(* CoDeSys 2.3 library: WagoLibODP_05.lib *)
(* Libraries: SerComm.lib 27.8.09 11:23:02, Serial_Interface_01.lib 1.2.10 12:53:52, SysLibRtc.lib 5.10.04 10:37:42, SysLibTime.lib 5.10.04 10:39:34, mod_com.lib 17.5.05 08:45:18, Standard.lib 22.11.04 11:21:12, SYSLIBCALLBACK.LIB 20.4.05 11:04:48 *)

(* Global variable list: Globale_Konstanten *)
VAR_GLOBAL CONSTANT
	gcODP_uiBUFFER_SIZE :	UINT := 65000; (* Absolut size of modbus buffer 'gODP_awData' *)

	gcODP_uiOFFSET_ONLINEREAD : UINT := 2000; (* Absolut startindex of OnlineReadArea in modbus buffer 'gODP_awData' *)
	gcODP_uiOFFSET_ONLINEWRITE: UINT := 2100; (* Absolut startindex of OnlineWriteArea in modbus buffer 'gODP_awData' *)
	gcODP_uiOFFSET_ALARM: UINT := 60000; 	  (* Absolut startindex of AlarmData in modbus buffer 'gODP_awData' *)

	gcODP_uiOFFSET_HISTORY_BASE: UINT := 4000; (* Absolut startindex of HistoryData in modbus buffer 'gODP_awData' *)
 	gcODP_uiHISTORY_ITEM_SIZE  : UINT := 2000; (* Offest for each iHistoryItem in modbus buffer 'gODP_awData' *)
 	gcODP_uiHISTORY_ITEM_COUNT : UINT := 1440; (* Number of entries for each iHistoryItem to store actual values in modbus buffer 'gODP_awData' *)

	gcODP_uiMAXVAR_ONLINEREAD : UINT := 100; 	(* Maximum number of variables in 'gODP_asConfigRead'*)
	gcODP_uiMAXVAR_ONLINEWRITE: UINT := 100; 	(* Maximum number of variables in 'gODP_asConfigWrite'*)
	gcODP_uiMAXVAR_HISTORY 	  : UINT := 100; 	(* Maximum number of variables in 'gODP_asConfigHistory'*)

	gcODP_uiMAXVAR_ALARMS 	  : UINT := 128; 	(* Maximum number of variables in 'gODP_asConfigAlarms'*)
	gcODP_uiSIZE_COMPRESSEDALARMS : UINT := 8; 	(* Size of compressed representation of all alarms in (gcODP_uiMAXVAR_ALARMS/16) *)

	gcODP_uiMAXALARMLOGENTRIES: UINT := 256; 	(* Maximum number of alarm entries in 'grODP_asAlarmLog'*)

	gcODP_bMODBUS_SLAVE_ID: BYTE := 1; (* Slave-ID for ODP-Online-Data and ODP-Historical values *)
	gcODP_bMODBUS_ALARM_SLAVE_ID: BYTE := 10;  (* Slave-ID for ODP-Alarm's  *)

	gcODP_tALARMRESPONSETIMEOUT: TIME := t#30s; (* Timeout for no response received from ODP-Server *)
	gcODP_tALARMINTERVALLINIT: TIME := t#2s; (* Initial intervall for retransmission of alarms *)
END_VAR

VAR_GLOBAL
	gODP_awData : ARRAY [0..gcODP_uiBUFFER_SIZE] OF WORD; (* The central ModbusBuffer *)

	gODP_asConfigRead 	: ARRAY [0..gcODP_uiMAXVAR_ONLINEREAD] OF tODP_Config;  (* Config data for each online read variable *)
	gODP_iCountOnlineReadVars 	: INT; (* Number of configuared tags in OnlineReadArea *)
	gODP_tOnlineIntervall : TIME := t#15s; (* Intervall to update the OnlineReadArea *)

	gODP_asConfigWrite 	: ARRAY [0..gcODP_uiMAXVAR_ONLINEWRITE] OF tODP_Config; (* Config data for each online write variable *)
	gODP_iCountOnlineWriteVars	: INT; (* Number of configuared tags in OnlineWriteArea *)

	gODP_asConfigHistory: ARRAY [0..gcODP_uiMAXVAR_HISTORY] OF tODP_Config;     (* Config data for each historical variable *)
	gODP_iCountHistoryVars	: INT; (* Number of configuared tags in HistoryArea *)

	gODP_asConfigAlarms : ARRAY [0..gcODP_uiMAXVAR_ALARMS] OF tODP_Alarm;    (* Config data for each alarm variable *)
	gODP_iCountAlarms	: INT; (* Number of configuared vars in AlarmArea *)
	gODP_awCompressedAlarms	: ARRAY [0..gcODP_uiSIZE_COMPRESSEDALARMS] OF WORD; (* Compressed (bitcoded) reprasentation of all alarms *)
	gODP_tAlarmIntervall: TIME := gcODP_tALARMINTERVALLINIT; (* Current intervall for retransmission of alarms *)
END_VAR

VAR_GLOBAL RETAIN
	(* Internal "Tag" based log for the last alarms *)
	grODP_uiAlarmLogIndex : UINT; (* Position in ring buffer of the last detected alarm *)
	grODP_asAlarmLog : ARRAY [0..gcODP_uiMAXALARMLOGENTRIES] OF tODP_AlarmLog; (* Ring buffer to the last alarms *)

	(* Sendbuffer for bitcoded(compressed) alarms *)
	grODP_asAlarmSendBuffer : ARRAY [0..gcODP_uiMAXALARMLOGENTRIES] OF tODP_AlarmBuffer; (* Ring buffer of compressed alarms *)
	grODP_uiCurrentAlarms : UINT; (* In specification called "Alarmzeiger" *)
	grODP_uiTransmittedAlarms : UINT; (* In specification called "Sendezeiger" *)

	grODP_uiAlarmIncrementor : UINT; (* Used as startaddress in alarm telegrams (ODP specific feature) *)
END_VAR

(* Data type *)
TYPE tODP_Alarm :
  STRUCT
	sTagName 	: STRING(12); 		(* TagName, displayed in ODP-Config *)
	iTagId	 	: INT;		 		(* TagId of alarm, given in 'ODP_RegisterTag()' *)
	dwAddress	: DWORD; 			(* Address of variable that should be monitored *)
	wMbWordIdx 	: WORD; 			(* ModbusAddress: Position in ODP data array 'awOdpData'. Descreipted as "KENNUNG" in  ODP-Specification Values: 0..999 *)
	bMbBitIdx	: BYTE;		 		(* ModbusAddress: Position of this Alarm in 'wMbWordIdx'. Values: 0..15 *)
	eAlarmState	: tODP_AlarmState;	(* State: Comming, ACK, Going *)
	xOldValue 	: BOOL;				(* Store the last value *)
  END_STRUCT
END_TYPE

(* Data type *)
TYPE tODP_AlarmBuffer :
STRUCT
	awCompressedAlarms : ARRAY [0..gcODP_uiSIZE_COMPRESSEDALARMS] OF WORD; (* bitcoded representation of all alarms *)
	tTime 			   : tODP_Time;		(* Current time of event *)
END_STRUCT
END_TYPE

(* Data type *)
TYPE tODP_AlarmLog :
  STRUCT
	iTagId	 	: INT;		 		(* TagId of alarm, given in 'ODP_RegisterTag()' *)
	eAlarmState	: tODP_AlarmState;	(* State: Comming, ACK, Going *)
	tTime 		: tODP_Time;		(* Current time of event *)
  END_STRUCT
END_TYPE

(* Data type *)
TYPE tODP_AlarmState :
(
	eOdpAlarmNONE 	:= 0,  (* unknown *)
	eOdpAlarmCOME 	:= 1,  (* A new alarm has been detected *)
	eOdpAlarmACK 	:= 2,  (* Alarm successful send to PC-Software "ODP-Config" *)
	eOdpAlarmGONE 	:= 3   (* Alarm is gone *)
);
END_TYPE

(* Data type *)
TYPE tODP_Config :
  STRUCT
	sTagName : STRING(12); 		(* TagName, displayed in ODP-Config *)
	dwAddress: DWORD; 			(* Address of variable that should be monitored  *)
	eDataType: tODP_DataType;	(* Datatype of variable *)
	wIndex	 : WORD; 			(* Position in ODP data array 'awOdpData' *)
  END_STRUCT
END_TYPE

(* Data type *)
TYPE tODP_DataType :
(
	eOdpTypeBOOL 	:= 1,
	eOdpTypeCHAR 	:= 2,
	eOdpTypeINT8 	:= 3,
	eOdpTypeUINT8 	:= 4,
	eOdpTypeINT16 	:= 5,
	eOdpTypeUINT16 	:= 6,
	eOdpTypeINT32 	:= 7,
	eOdpTypeUINT32 	:= 8,
	eOdpTypeINT64 	:= 9,
	eOdpTypeUINT64 	:= 10,
	eOdpTypeFLOAT32 := 11,
	eOdpTypeFLOAT64 := 12,
	eOdpTypeSTRING 	:= 13,
	eOdpTypeBLOB 	:= 14
);
END_TYPE

(* Data type *)
TYPE tODP_Table :
(
	eOdpTableRead 	:= 1,
	eOdpTableWrite	:= 2,
	eOdpTableHistory:= 3,
	eOdpTableAlarm	:= 4
);
END_TYPE

(* Data type *)
TYPE tODP_Time :
  STRUCT
	bMinute : BYTE;
	bSecond : BYTE;
	bDay 	: BYTE;
	bHour 	: BYTE;
   	bYear 	: BYTE; (* Based on Year 1970 *)
	bMonth 	: BYTE;
  END_STRUCT
END_TYPE

(* POU PLC_PRG, ST *)
PROGRAM PLC_PRG
VAR
	(* ODP-Config Flag *)
	xODPInitDone : BOOL := FALSE;

	(* ODP variables to ODP-Config *)
	wReadVar_01 : WORD;
	iReadVar_02 : INT;
	uiReadVar_03: UINT;
	wMyPT100_Ch2 AT %IW1: WORD; (* Channel 2 of first analog input *)
	xMyFirstDI AT %IX2.0 : BOOL; (* Could not be monitored directly - must be mapped to helper*)
	wMyFirstDI : WORD; 	(* ODP helper variable for boolean process data *)

	(* ODP variables from ODP-Config *)
	wWriteVar_01 : WORD;
	iWriteVar_02 : INT;
	uiWriteVar_03: UINT;

	(* ODP error, alarms and messages *)
	xError_01 : BOOL; (* F1: 400V PowerSupply fails *)
	xError_02 : BOOL; (* Material buffer is empty   *)
	xError_03 : BOOL;
	xAlarm_01 : BOOL; (* Temperatur xy to high *)
	xAlarm_02 : BOOL;
	xAlarm_03 : BOOL;
	xMsg_01   : BOOL; (* Mode: "auto" -> "manual"  *)
	xMsg_02   : BOOL; (* Mode: "manual" -> "auto"  *)
	xMsg_03   : BOOL; (* Recepies: Load new        *)
	(* ModbusCommunication *)
	xConnected : BOOL;
	dwRequestCount:DWORD;
	dtLastRequest:DT;
	dwAlarmsCurrent:DWORD;
	dwAlarmsTransmitted:DWORD;
	dtLastTransmittedAlarm:DT;

END_VAR
(* Produce monitoring data *)
wReadVar_01 := wReadVar_01 +1;
iReadVar_02 := iReadVar_02 -2;
uiReadVar_03:= uiReadVar_03 +3;

(* Map boolean processdata on helper variable *)
wMyFirstDI := BOOL_TO_WORD(xMyFirstDI);

(* Start Modbus communication *)
ODP_AGENT(	EN:= TRUE,
			bCOM_PORT:= 0,		(* 0:= 873 Onboard; 1:= ServicePort; 2...n:= additional RS232 Modules 750-650 *)
			cbCOM_BAUDRATE:= BAUD_9600,
			cpCOM_PARITY:= PARITY_NO,
			csCOM_STOPBITS:= STOPBITS_1,
			cbsCOM_BYTESIZE:= BS_8,
			cfCOM_FLOW_CONTROL:= NO_FLOW_CONTROL, (* RTS_CTS; NO_FLOW_CONTROL *)
			xConnected => xConnected,
			dwRequestCount=> dwRequestCount,
			dtLastRequest=> dtLastRequest,
			dwAlarmsCurrent=> dwAlarmsCurrent,
			dwAlarmsTransmitted=> dwAlarmsTransmitted,
			dtLastTransmittedAlarm=> dtLastTransmittedAlarm);

(* Config ODP-Server *)
IF NOT xODPInitDone THEN
	(* Init ODP-Configblock *)
	ODP_InitOdpConfig('MyODPLogger', t#15s);
	(* Register variables of OnlineReadArea *)
	ODP_RegisterTag(eOdpTableRead, 'wReadVar_01', ADR(PLC_PRG.wReadVar_01), eOdpTypeUINT16);
	ODP_RegisterTag(eOdpTableRead, 'iReadVar_02', ADR(PLC_PRG.iReadVar_02), eOdpTypeINT16);
	ODP_RegisterTag(eOdpTableRead, 'uiReadVar_03', ADR(PLC_PRG.uiReadVar_03), eOdpTypeUINT16);
	ODP_RegisterTag(eOdpTableRead, 'myPT100_CH2', ADR(PLC_PRG.wMyPT100_Ch2), eOdpTypeUINT16);
	ODP_RegisterTag(eOdpTableRead, 'wMyFirstDI', ADR(PLC_PRG.wMyFirstDI), eOdpTypeUINT16);
	(* Register variables of OnlineWriteArea *)
	ODP_RegisterTag(eOdpTableWrite, 'wWriteVar_01', ADR(PLC_PRG.wWriteVar_01), eOdpTypeUINT16);
	ODP_RegisterTag(eOdpTableWrite, 'iWriteVar_02', ADR(PLC_PRG.iWriteVar_02), eOdpTypeINT16);
	ODP_RegisterTag(eOdpTableWrite, 'uiWriteVar_03', ADR(PLC_PRG.uiWriteVar_03), eOdpTypeUINT16);
	(* Register variables of HistoryArea *)
	ODP_RegisterTag(eOdpTableHistory, 'wReadVar_01', ADR(PLC_PRG.wReadVar_01), eOdpTypeUINT16);
	ODP_RegisterTag(eOdpTableHistory, 'iReadVar_02', ADR(PLC_PRG.iReadVar_02), eOdpTypeINT16);
	(* Register Alarm(SAM's) *)
	ODP_RegisterTag(eOdpTableAlarm, 'xError_01', ADR(PLC_PRG.xError_01), eOdpTypeBOOL);
	ODP_RegisterTag(eOdpTableAlarm, 'xError_02', ADR(PLC_PRG.xError_02), eOdpTypeBOOL);
	ODP_RegisterTag(eOdpTableAlarm, 'xError_03', ADR(PLC_PRG.xError_03), eOdpTypeBOOL);
	ODP_RegisterTag(eOdpTableAlarm, 'xAlarm_01', ADR(PLC_PRG.xAlarm_01), eOdpTypeBOOL);
	ODP_RegisterTag(eOdpTableAlarm, 'xAlarm_02', ADR(PLC_PRG.xAlarm_02), eOdpTypeBOOL);
	ODP_RegisterTag(eOdpTableAlarm, 'xAlarm_03', ADR(PLC_PRG.xAlarm_03), eOdpTypeBOOL);
	ODP_RegisterTag(eOdpTableAlarm, 'xMsg_01', ADR(PLC_PRG.xMsg_01), eOdpTypeBOOL);
	ODP_RegisterTag(eOdpTableAlarm, 'xMsg_02', ADR(PLC_PRG.xMsg_02), eOdpTypeBOOL);
	ODP_RegisterTag(eOdpTableAlarm, 'xMsg_03', ADR(PLC_PRG.xMsg_03), eOdpTypeBOOL);
	xODPInitDone := TRUE;
END_IF
END_PROGRAM

(* POU ODP_AGENT, ST *)
PROGRAM ODP_AGENT
(* This program work as conterpart for datalogger "ODP" from company VIDEC.
It waits for ODP-Request on serial port (Modbus_RTU).
In addition this program can send alarm telegrams.
*)
VAR_INPUT
	EN					:	BOOL := TRUE;
	bCOM_PORT			:	BYTE				:= 0; (* RS232 OnBoard 750-873 *)
	cbCOM_BAUDRATE		:	COM_BAUDRATE 		:= BAUD_9600;
	cpCOM_PARITY		:	COM_PARITY 			:= PARITY_NO;
	csCOM_STOPBITS		:	COM_STOPBITS 		:= STOPBITS_1;
	cbsCOM_BYTESIZE		:	COM_BYTESIZE 		:= BS_8;
	cfCOM_FLOW_CONTROL	:	COM_FLOW_CONTROL 	:= NO_FLOW_CONTROL ;
END_VAR
VAR_OUTPUT
	(* Online/Historic-Data*)
	xConnected :	BOOL; (* ODP-Server is connected *)
	dwRequestCount: DWORD; (* Number of received Modbus-Requests from ODP-Server *)
	dtLastRequest : DT; (* Timestamp of last received modbus request from ODP-Server*)
	(* Alarms *)
	dwAlarmsCurrent : DWORD; (* Number of local detected alarms  *)
	dwAlarmsTransmitted : DWORD; (* Number of transmitted alarms *)
	dtLastTransmittedAlarm : DT; (* Timestamp of last succesful tranmitted alarm *)
END_VAR
VAR
	(* ODP --------------------------------*)
	tCurTime 	: tODP_Time;

	xUpdateOdpWriteAreaRequired : BOOL; (* Update WriteArea after each modbus write access *)
	oTonRead 	: TON; (* Timer to update ReadArea with fresh values *)

	xSendAlarm	: BOOL; (* Flag to send an alarm to PC-Software "ODP-Config". Reset after receiving succesful acknoledge *)
	oTonAlarmResponseTimeout : TON; (* Timer to check if server acknoledge alarm within given time *)
	oTonAlarmIntervall	: TON; (* ODP: Intervall timer for minimal gap between two alarm telegrams *)

	(* ODP-Historic data *)
	bLastMinute : BYTE; (* Used to implement the intervall for writing historical data *)
	wState : WORD; (* Used in statemashiene to clear all historical data in seperate plc cycles *)
	uiCurrent : UINT; (* Index of a historical variable, used to iterate along all historical variables *)

	(* Modbus WatchDog ---------------------*)
	oTonWatchDog : TON; (* Timer to check if PC-Software "ODP-Config" is connected *)


	(* Serial-Interface --------------------*)
	oComPort		: SERIAL_INTERFACE;
	ReceiveBuffer	: typRING_BUFFER;
	RecBufferSize   : INT; (* Size member 'data' of bytes  *)
	abSendBuffer	: ARRAY[0..512] OF BYTE;
	iBytesToSend	: INT;  (* Number of bytes that should be send *)
	SendActive		: BOOL;
	xSendActiveOld  : BOOL;
	xReset			: BOOL;
	RecBufferOldIdx	: INT; (* Begin of next telegram in ringbuffer *)
	helpIdx 		: INT;
	iTo				: INT; (* Number of bytes to process *)
	oTonSendWait 	: TON; (* Detect falling edge of xSendActive and wait to make shure all data are transmitted *)
	xSendWait 		: BOOL;

	(* Local-Modbus-Slave -------------------*)
	SlaveId			: BYTE; (* received SlaveAddress from remote modbus master *)
	FunctionCode	: BYTE; (* received FunctionCode from remote modbus master *)
	UnitId			: BYTE;
	StartAddress	: WORD;
	NumberOfPoints	: WORD;

	LocalByte		: BYTE;
	BitCount		: BYTE;
	Mask			: BYTE;

	xSendResponse	: BOOL;
	ErrorCode		: BYTE;

	xIllegalFunctionCode: BOOL; (* Flag: Indicates the receiving of an unsupported or unknown FunctionCode *)

	abSlaveResponse	: ARRAY[0..512] OF BYTE; (* Buffer to build the response of the local Modbus-Slave *)
	iSlaveResponseLength: INT; (* Number of bytes that should be send *)
	iSlaveRequestLength : INT; (* Length of received bytes *)

	(* Local-Modbus-Master-----------------*)
	abMasterRequest		: ARRAY[0..125] OF BYTE; (* Buffer to build the Request of the local Modbus-Master *)
	xSendRequest		: BOOL; (* Flag to send one modbus-request to PC-Software "ODP-Config". Reset direct after transmission *)
	abMasterResponse	: ARRAY[0..19] OF BYTE; (* Buffer to process the Response from the remote Modbus-Master *)

	(* CRC16 Check ------------------------*)
	CALC_CRC			:	CRC16;  (* Function block to calculate CRC16 *)
	CRC_RTU				:	WORD;

	(* Little Helpers ---------------------*)
	i	: 	INT;
	wHelp :	WORD; (* *)

END_VAR
(* ODP: Get current time from RTC *)
tCurTime := ODP_GetTime(); (* Read current time from RTC *)

(* Update ODP-Config block (at index 8) each cycle *)
ODP_UpdateConfigArea(); (* Also update local RTC, when requested by PC-Software "ODP-Config" indicated by TRUE (at index 17) *)

(* Clear all historical data if requested *)
CASE wState OF
0: (* IDLE - Wait for something to do *)
	IF gODP_awData[37] = 16#0001 THEN
		uiCurrent := 0; (* Set Index to the first HistVar *)
		wState := 10; (* Go Ahead *)
	END_IF

10: (* Check if all historical data are reset to "INVALID_VALUE" *)
	IF uiCurrent < gODP_iCountHistoryVars THEN
		(* There are more HistVars to reset *)
		wState := 20; (* Go Ahead *)
	ELSE
		(* All HistVars are reseted *)
		gODP_awData[37] := 16#0000;
		wState := 0; (* Done *)
	END_IF

20: (* Overwrite all historical data of current HistVar with "INVALID_VALUE" *)
	FOR i:=0 TO gcODP_uiHISTORY_ITEM_COUNT-1 DO
		gODP_awData[gODP_asConfigHistory[uiCurrent].wIndex] := gODP_awData[36];
	END_FOR
	(* Set index to next HistVar *)
	uiCurrent := uiCurrent +1;
	wState := 10; (* Go Ahead *)
END_CASE

(* Check current values of all configurated alarms *)
ODP_CheckAlarms(tCurTime);

(* Check if an alarm have to be send to PC-Software "ODP-Config" *)
(* ODP: Intervall timer for minimal gap between two alarm telegrams *)
oTonAlarmIntervall(IN:=(NOT xSendAlarm), PT:= gODP_tAlarmIntervall);
IF oTonAlarmIntervall.Q THEN
	IF grODP_uiCurrentAlarms <> grODP_uiTransmittedAlarms THEN
		(* ALARM DETECTED: Send modbus request to PC-Software "ODP-Config" *)
		xSendAlarm := TRUE; (* Flag to send an alarm to PC-Software "ODP-Config". Reset after receiving succesful acknoledge *)
		xSendRequest := TRUE; (* Flag to send one modbus-request to PC-Software "ODP-Config". Reset direct after transmission *)
	END_IF
END_IF

(* Check if ODP-Server acknoledge alarm within given timeout *)
oTonAlarmResponseTimeout(IN:=xSendAlarm, PT:=gcODP_tALARMRESPONSETIMEOUT);
IF oTonAlarmResponseTimeout.Q THEN
	(* We do not receive the alarm acknoledge *)
	oTonAlarmResponseTimeout(IN:=FALSE); (* Reset timer *)
	gODP_tAlarmIntervall := gODP_tAlarmIntervall * 2; (* Increment retransmission intervall by factor 2 *)
	xSendAlarm := FALSE;
END_IF

(* Copy to output *)
dwAlarmsCurrent := grODP_uiCurrentAlarms;
dwAlarmsTransmitted := grODP_uiTransmittedAlarms;

(* ODP: Update historical data area*)
IF tCurTime.bMinute <> bLastMinute THEN
	bLastMinute := tCurTime.bMinute;
	ODP_UpdateHistory(tCurTime); (* Write current values to history *)
END_IF

(* ODP: Update OnlineWriteArea after each modbus write access *)
IF xUpdateOdpWriteAreaRequired THEN
	xUpdateOdpWriteAreaRequired := FALSE;
	ODP_UpdateOnlineWriteArea();
END_IF

(* ODP: Update OnlineReadArea with fresh values *)
oTonRead(IN:=TRUE, PT:= gODP_tOnlineIntervall);
IF oTonRead.Q THEN
	oTonRead(IN:=FALSE);
	ODP_UpdateOnlineReadArea();
END_IF

(* ODP: WatchDog to check connection with remote modbus master  *)
oTonWatchDog(IN:=TRUE, PT:= (gODP_tOnlineIntervall *8));
IF oTonWatchDog.Q THEN
	xConnected:= FALSE;
END_IF

(* Serial-Interface: Main -----------------------------*)
oComPort(	xOPEN_COM_PORT 	:= EN,
			bCOM_PORT_NR	:= bCOM_PORT,
			cbBAUDRATE		:= cbCOM_BAUDRATE,
			cpPARITY		:= cpCOM_PARITY,
			csSTOPBITS		:= csCOM_STOPBITS,
			cbsBYTESIZE		:= cbsCOM_BYTESIZE,
			cfFLOW_CONTROL	:= cfCOM_FLOW_CONTROL,
			iBYTES_TO_SEND	:= iBytesToSend,
			ptSEND_BUFFER	:= ADR(abSendBuffer[0]),
			xSTART_SEND		:= SendActive,
			utRECEIVE_BUFFER:= ReceiveBuffer,
			xINIT			:= xReset);

(* Detect falling edge of SendActive and wait to make shure all data are transmitted *)
IF (NOT SendActive) AND xSendActiveOld THEN
	oTonSendWait(IN:=FALSE);
END_IF
xSendActiveOld := SendActive;
oTonSendWait(IN:=TRUE , PT:= t#50ms);

IF (NOT SendActive) AND (oTonSendWait.Q) THEN
	(* Serial-Interface: Check ReceiveBuffer for something to do ------*)
	IF ReceiveBuffer.Index <> RecBufferOldIdx THEN
		RecBufferSize := SIZEOF(ReceiveBuffer.Data);
		(* Calculate number of received bytes  *)
		iTo	:= ReceiveBuffer.Index - RecBufferOldIdx ;
		(* Check if telegram exceed border of ringbuffer *)
		IF iTo < 0 THEN
			iTo := iTo + RecBufferSize;
		END_IF;
		(* Check if minimal telegram length is received *)
		IF iTo <= 4 THEN
			(************************************************************)
			RETURN;(*******  MINIMAL TELEGRAM LENGTH NOT REACHED ********)
			(************************************************************)
		ELSE (* iTo <= 4 *)
			(* Check Modbus-Slave-Address to obtain if telegram is a 'Modbus-Slave-Response' or a 'Modbus-Master-Request' *)
			SlaveId := ReceiveBuffer.Data[RecBufferOldIdx]; (* store Slaveaddress *)
			FunctionCode := ReceiveBuffer.Data[(RecBufferOldIdx+1) MOD RecBufferSize];	(* store FunctionCode *)

			IF SlaveId = gcODP_bMODBUS_ALARM_SLAVE_ID THEN (* -----  Telegram is a Modbus-Slave-Response  ------------------------*)
				(* Check Exceptionbit in field "FUNCTIONCODE" is set to recognise if successful or not *)
				IF ( FunctionCode AND 16#80) <> 0 THEN
					(* Sending "Alarm" to ODP-Server fails - retransmission is done by timeout *)
					RecBufferOldIdx := (RecBufferOldIdx +5) MOD RecBufferSize; (* Length of modbus execption telegram *)
					(* Reset flag for send alarm to ODP-Server *)
					xSendAlarm := FALSE;
					(* Increment Sendezeiger *)
					grODP_uiTransmittedAlarms := (grODP_uiTransmittedAlarms +1) MOD gcODP_uiMAXALARMLOGENTRIES;
				ELSE (* ( FunctionCode AND 16#80) <> 0 *)
					(* Sending "Alarm" to ODP-Server successful executed *)
					IF iTo >=8 THEN (* Wait until complied telegram of 8 bytes received *)
						(* Copy telegram data into 'abMasterResponse'*)
						FOR i:=0 TO iTo DO
							helpIdx := (RecBufferOldIdx + i) MOD RecBufferSize;
							abMasterResponse[i] :=  ReceiveBuffer.Data[ helpIdx ];
						END_FOR;
						(* Alarm successful transmitted, mark Alarm job as done in alarmlog *)
						ODP_UpdateAlarmLog(	0,
											eOdpAlarmACK,
											tCurTime);
						(* Set alarm transfer intervall to initial time *)
			    		gODP_tAlarmIntervall := gcODP_tALARMINTERVALLINIT;
						(* Set readpointer to the next modbus header *)
						RecBufferOldIdx := (RecBufferOldIdx +8) MOD RecBufferSize;
						(* Reset flag for send alarm to ODP-Server *)
						xSendAlarm := FALSE;
						(* Increment Sendezeiger *)
						grODP_uiTransmittedAlarms := (grODP_uiTransmittedAlarms +1) MOD gcODP_uiMAXALARMLOGENTRIES;
						dtLastTransmittedAlarm := SysRtcGetTime(TRUE);
					END_IF;
				END_IF

			ELSE (* ----- Telegram is a Modbus-Master-Request -------------------------------------------------*)
				(* Check FunctionCode *)
				CASE Functioncode OF

				16#03, (* FC3: Read Holding Registers 	*)
				16#04: (* FC4: Read Input Registers 	*)
					iSlaveRequestLength := 8;
					IF iTo >= iSlaveRequestLength THEN
						(* Check SlaveId against local SlaveAddress *)
						IF SlaveId <> gcODP_bMODBUS_SLAVE_ID THEN
							(* Ignore received telegram, just set readpointer to the next modbus header *)
							RecBufferOldIdx := (RecBufferOldIdx +iSlaveRequestLength) MOD RecBufferSize;
						ELSE
							(* Calculate CRC of modbus request from remote modbus master *)
							CALC_CRC(INPUT:=16#00, EN:=FALSE);
							FOR i := 0 TO 5 DO
								CALC_CRC(INPUT:=ReceiveBuffer.Data[(RecBufferOldIdx +i) MOD RecBufferSize], EN:=TRUE);
							END_FOR
							CRC_RTU := (ReceiveBuffer.Data[(RecBufferOldIdx+6) MOD RecBufferSize] * 16#0100)
										OR ReceiveBuffer.Data[(RecBufferOldIdx+7) MOD RecBufferSize];
							(* Check CRC *)
							IF CRC_RTU <> CALC_CRC.CRC THEN
								(* Send modbusexecption response to remote modbus master *)
								abSlaveResponse[0]:= SlaveId;  				(* Copy Slaveaddress into response *)
								abSlaveResponse[1]:= FunctionCode OR 16#80;	(* Copy FunctionCode into response and set ExceptionFlag*)
								abSlaveResponse[2]:= 16#03;	 				(* ILLEGAL DATA VALUE *)
								iSlaveResponseLength := 3;
								xSendResponse := TRUE; (***********************************)
							ELSE
								StartAddress := (ReceiveBuffer.Data[(RecBufferOldIdx+2)MOD RecBufferSize] * 16#0100)
												OR ReceiveBuffer.Data[(RecBufferOldIdx+3)MOD RecBufferSize];
								NumberOfPoints := (ReceiveBuffer.Data[(RecBufferOldIdx+4)MOD RecBufferSize] * 16#0100)
												OR ReceiveBuffer.Data[(RecBufferOldIdx+5)MOD RecBufferSize];
								(* Check modbus start address *)
								IF (StartAddress + NumberOfPoints) >= (SIZEOF(gODP_awData) /2) THEN
									(* Send modbusexecption response to remote modbus master *)
									abSlaveResponse[0]:= SlaveId;  				(* Copy SlaveAddress into response *)
									abSlaveResponse[1]:= FunctionCode OR 16#80;	(* Copy FunctionCode into response and set ExceptionFlag*)
									abSlaveResponse[2]:= 16#02;	  				(* ILLEGAL DATA ADDRESS *)
									iSlaveResponseLength := 3;
									xSendResponse := TRUE; (***********************************)
								ELSE
									(* Receiving a valid modbus request from remote master *)
									abSlaveResponse[0]:= SlaveId;  		(* Copy SlaveAddress into response *)
									abSlaveResponse[1]:= FunctionCode;	(* Copy FunctionCode into response *)
									abSlaveResponse[2]:= WORD_TO_BYTE(NumberOfPoints*2); (* Number of bytes *)
									(* Copy data into response *)
									FOR i:=0 TO NumberOfPoints-1 DO
										abSlaveResponse[4+(2*i)] := WORD_TO_BYTE(gODP_awData[StartAddress +i]);
										abSlaveResponse[3+(2*i)] := WORD_TO_BYTE(SHR(gODP_awData[StartAddress +i],8));
									END_FOR;
									iSlaveResponseLength := (NumberOfPoints*2)+3;
									xSendResponse := TRUE; (***********************************)
									(* Reset connection watch dog *)
									oTonWatchDog(IN:=FALSE); (* Reset WatchDog *)
									xConnected := TRUE;
									dwRequestCount := dwRequestCount +1;
									dtLastRequest := SysRtcGetTime(TRUE);
								END_IF (* (StartAddress + NumberOfPoints) >= (SIZEOF(gODP_awData) /2) *)
							END_IF (* CRC_RTU <> CALC_CRC.CRC *)
						END_IF (* SlaveId <> gcODP_bMODBUS_SLAVE_ID *)
					END_IF (* iTo >= iSlaveRequestLength *)

				16#10 : (* FC16: Preset Multible Registers	*)
					IF iTo >= 6 THEN
						(* Calculate Requestlength *)
						NumberOfPoints := (ReceiveBuffer.Data[(RecBufferOldIdx+4) MOD RecBufferSize] * 16#0100)
										OR ReceiveBuffer.Data[(RecBufferOldIdx+5) MOD RecBufferSize];
						iSlaveRequestLength := ReceiveBuffer.Data[(RecBufferOldIdx+6) MOD RecBufferSize] +9;
						IF iTo >= iSlaveRequestLength THEN (* All bytes received? *)
							(* Check SlaveId against local SlaveAddress *)
							IF SlaveId <> gcODP_bMODBUS_SLAVE_ID THEN
								(* Ignore received telegram, just set writepointer to the next modbus header *)
								RecBufferOldIdx := (RecBufferOldIdx +iSlaveRequestLength) MOD RecBufferSize;
							ELSE (* SlaveId <> gcODP_bMODBUS_SLAVE_ID *)
								(* Calculate CRC from Received Message *)
								CALC_CRC(INPUT:=16#00, EN:=FALSE);
								FOR i:=0 TO iSlaveRequestLength-3 DO
									CALC_CRC(INPUT:=ReceiveBuffer.Data[(RecBufferOldIdx+i) MOD RecBufferSize], EN:=TRUE);
								END_FOR
								CRC_RTU := (ReceiveBuffer.Data[(RecBufferOldIdx+iSlaveRequestLength-2) MOD RecBufferSize] * 16#0100)
											OR ReceiveBuffer.Data[(RecBufferOldIdx+iSlaveRequestLength-1) MOD RecBufferSize];
								(* Check CRC *)
								IF CRC_RTU <> CALC_CRC.CRC THEN
									(* Send modbusexecption response to remote modbus master *)
									abSlaveResponse[0]:= SlaveId;  				(* Copy Slaveaddress into response *)
									abSlaveResponse[1]:= FunctionCode OR 16#80;	(* Copy FunctionCode into response and set ExceptionFlag*)
									abSlaveResponse[2]:= 16#03;	 				(* ILLEGAL DATA VALUE *)
									iSlaveResponseLength := 3;
									xSendResponse := TRUE; (***********************************)
								ELSE
									StartAddress := (ReceiveBuffer.Data[(RecBufferOldIdx+2)MOD RecBufferSize] * 16#0100)
												OR ReceiveBuffer.Data[(RecBufferOldIdx+3)MOD RecBufferSize];
									(* Check modbus start address *)
									IF (StartAddress + NumberOfPoints) >= (SIZEOF(gODP_awData) /2) THEN
										(* Send modbusexecption response to remote modbus master *)
										abSlaveResponse[0]:= SlaveId;  				(* Copy SlaveAddress into response *)
										abSlaveResponse[1]:= FunctionCode OR 16#80;	(* Copy FunctionCode into response and set ExceptionFlag*)
										abSlaveResponse[2]:= 16#02;	  				(* ILLEGAL DATA ADDRESS *)
										iSlaveResponseLength := 3;
										xSendResponse := TRUE; (***********************************)
									ELSE
										(* Accept received data *)
										FOR i:=0 TO NumberOfPoints-1 DO
											gODP_awData[StartAddress +i] := (ReceiveBuffer.Data[(RecBufferOldIdx+7+(2*i))MOD RecBufferSize] * 16#0100)
																	OR ReceiveBuffer.Data[(RecBufferOldIdx+8+(2*i))MOD RecBufferSize];
										END_FOR
										(* Send positive modbus response to remote modbus master *)
										abSlaveResponse[0]:= SlaveId;  							 (* Copy SlaveAddress into response *)
										abSlaveResponse[1]:= FunctionCode;						 (* Copy FunctionCode into response and set ExceptionFlag*)
										abSlaveResponse[2]:= WORD_TO_BYTE(SHR(StartAddress,8));	 (* Startaddress Hi*)
										abSlaveResponse[3]:= WORD_TO_BYTE(StartAddress);	  	 (* Startaddress Lo*)
										abSlaveResponse[4]:= WORD_TO_BYTE(SHR(NumberOfPoints,8));(* Number of words written Hi*)
										abSlaveResponse[5]:= WORD_TO_BYTE(NumberOfPoints);		 (* Number of words written Lo*)
										iSlaveResponseLength := 6;
										xSendResponse := TRUE; (***********************************)
										(* Set Flag for write received data to local variables *)
										xUpdateOdpWriteAreaRequired := TRUE;
									END_IF (* (StartAddress + NumberOfPoints) >= (SIZEOF(gODP_awData) /2) *)
								END_IF (* CRC_RTU <> CALC_CRC.CRC *)
							END_IF (* SlaveId <> gcODP_bMODBUS_SLAVE_ID *)
						END_IF (* iTo >= iSlaveRequestLength *)
					END_IF (* iTo >= 6 *)

				ELSE (* Protocol error: Unexpected FUNCTIONCODE found in receive buffer *)
					xIllegalFunctionCode := TRUE;
					(* Check SlaveId against local SlaveAddress *)
					IF SlaveId <> gcODP_bMODBUS_SLAVE_ID THEN
						(* Ignore received telegram, and reset receive buffer, because absolute length of request are unknown *)
						RecBufferOldIdx := 0;
						ReceiveBuffer.Index := 0;
						FOR i:=0 TO (RecBufferSize-1) DO
							ReceiveBuffer.Data[i];
						END_FOR
					ELSE
						(* Send modbusexecption response to remote modbus master *)
						abSlaveResponse[0]:= SlaveId;  				(* Copy SlaveAddress into response *)
						abSlaveResponse[1]:= FunctionCode OR 16#80;	(* Copy FunctionCode into response and set ExceptionFlag*)
						abSlaveResponse[2]:= 16#01;	  				(* ILLEGAL FUNCTIONCODE *)
						iSlaveResponseLength := 3;
						xSendResponse := TRUE; (***********************************)
					END_IF
				END_CASE;
			END_IF
		END_IF (* iTo <= 4 *)
	END_IF (* ReceiveBuffer.Index <> RecBufferOldIdx *)


	IF xSendResponse THEN (* Send response to remote modbus master ------------------*)
		xSendResponse := FALSE;
		(* Calculate CRC for modbus response *)
		CALC_CRC(INPUT:=16#00, EN:=FALSE);
		FOR i := 0 TO (iSlaveResponseLength - 1) DO
			CALC_CRC(INPUT :=  abSlaveResponse[i], EN := TRUE);
		END_FOR;
		(* Append CRC to modbus response *)
		abSlaveResponse[iSlaveResponseLength ] := WORD_TO_BYTE(SHR(CALC_CRC.CRC,8));
		abSlaveResponse[iSlaveResponseLength + 1] := WORD_TO_BYTE(CALC_CRC.CRC);
		iSlaveResponseLength := iSlaveResponseLength + 2;
		(* Copy modbus response into sendbuffer *)
		FOR i := 0 TO (iSlaveResponseLength - 1) DO
			abSendBuffer[i] := abSlaveResponse[i];
		END_FOR
		iBytesToSend := iSlaveResponseLength;
		SendActive := TRUE; (*********************************)
		IF NOT xIllegalFunctionCode THEN
			(* Set RecBufferOldIdx to next modbus header *)
			RecBufferOldIdx := (RecBufferOldIdx + iSlaveRequestLength) MOD RecBufferSize;
		ELSE
			(* Reset receive buffer, because absolute length of request can not identified *)
			RecBufferOldIdx := 0;
			ReceiveBuffer.Index := 0;
			xIllegalFunctionCode := FALSE;
		END_IF
		RETURN;

	ELSIF xSendRequest THEN (* Send request to remote modbus slave ------------------*)
		xSendRequest := FALSE;
		(* Increment startaddress of alarm telegrams (ODP specific feature) *)
		grODP_uiAlarmIncrementor := grODP_uiAlarmIncrementor +1;
		(* Calculate index of the next alarm in grODP_asAlarmSendBuffer that should be transmitted *)
		wHelp := (grODP_uiTransmittedAlarms +1) MOD gcODP_uiMAXALARMLOGENTRIES;
		(* Build request telegram *)
		abSendBuffer[ 0] := gcODP_bMODBUS_ALARM_SLAVE_ID; (* Modbus-Slave Address of PC-Software "ODP-Config" *)
		abSendBuffer[ 1] := 16#10; (* FunctionCode 16: preset multiple registers *)
		abSendBuffer[ 2] := WORD_TO_BYTE(SHR(grODP_uiAlarmIncrementor,8)); (* Startaddress High *)
		abSendBuffer[ 3] := WORD_TO_BYTE(grODP_uiAlarmIncrementor); (* Startaddress Low *)
		abSendBuffer[ 4] := 16#00; 									(* Word count - High *)
		abSendBuffer[ 5] := 5 + gcODP_uiSIZE_COMPRESSEDALARMS;		(* Word count - Low *)
		abSendBuffer[ 6] := 2* abSendBuffer[5]; 					(* Byte count  *)
		(* Insert "Kennung"  *)
		abSendBuffer[ 7] := 16#00;
		abSendBuffer[ 8] := 16#00;
		(* Insert "Value" *)
		abSendBuffer[ 9] := 16#00;
		abSendBuffer[10] := 16#00;
		(* Insert "timestamp" *)
		abSendBuffer[11] := grODP_asAlarmSendBuffer[wHelp].tTime.bYear;
		abSendBuffer[12] := grODP_asAlarmSendBuffer[wHelp].tTime.bMonth;
		abSendBuffer[13] := grODP_asAlarmSendBuffer[wHelp].tTime.bDay;
		abSendBuffer[14] := grODP_asAlarmSendBuffer[wHelp].tTime.bHour;
		abSendBuffer[15] := grODP_asAlarmSendBuffer[wHelp].tTime.bMinute;
		abSendBuffer[16] := grODP_asAlarmSendBuffer[wHelp].tTime.bSecond;
		(* Insert compressed representation of all alarms *)
		FOR i:=0 TO (gcODP_uiSIZE_COMPRESSEDALARMS -1) DO
			abSendBuffer[17+(2*i)] := WORD_TO_BYTE(SHR(grODP_asAlarmSendBuffer[wHelp].awCompressedAlarms[i], 8)); (* Compressed (bitcoded) reprasentation of all alarms *)
			abSendBuffer[18+(2*i)] := WORD_TO_BYTE(grODP_asAlarmSendBuffer[wHelp].awCompressedAlarms[i]);         (* Compressed (bitcoded) reprasentation of all alarms *)
		END_FOR
		(*  Calculate CRC *)
		CALC_CRC(INPUT:=16#00, EN:=FALSE);
		FOR i := 0 TO (16 + (2*gcODP_uiSIZE_COMPRESSEDALARMS)) DO
			CALC_CRC(INPUT:=abSendBuffer[i], EN:=TRUE);
		END_FOR;
		(* Append CRC to modbus response *)
		abSendBuffer[17+(2*gcODP_uiSIZE_COMPRESSEDALARMS)] := WORD_TO_BYTE(SHR(CALC_CRC.CRC,8));
		abSendBuffer[18+(2*gcODP_uiSIZE_COMPRESSEDALARMS)] := WORD_TO_BYTE(CALC_CRC.CRC);
		(* Set "SendActive := TRUE; *)
		iBytesToSend := 19+(2*gcODP_uiSIZE_COMPRESSEDALARMS);
		SendActive := TRUE; (*********************************)
		RETURN;
	END_IF (* xSendResponse ELSIF xSendRequest*)

END_IF (* NOT SendActive *)
END_PROGRAM

(* POU ODP_GetTime, ST *)
FUNCTION ODP_GetTime : tODP_Time
(* This function read the current time from the RTC and convert it into tODP_Time format. *)
VAR_INPUT
END_VAR
VAR
	oCurTimeEx : CurTimeEx; (* Functionblock from SysLibTime *)
	SysTime: SysTime64;
	SysTD: SystemTimeDate;
END_VAR
oCurTimeEx(SystemTime:= SysTime, TimeDate:= SysTD );

ODP_GetTime.bSecond := UINT_TO_BYTE(SysTD.Second);
ODP_GetTime.bMinute := UINT_TO_BYTE(SysTD.Minute);
ODP_GetTime.bHour 	:= UINT_TO_BYTE(SysTD.Hour);
ODP_GetTime.bDay 	:= UINT_TO_BYTE(SysTD.Day);
ODP_GetTime.bMonth  := UINT_TO_BYTE(SysTD.Month);
IF SysTD.Year >= 2000 THEN
	ODP_GetTime.bYear  	:= UINT_TO_BYTE(SysTD.Year -2000);
ELSE
	ODP_GetTime.bYear  	:= 16#00;
END_IF
END_FUNCTION

(* POU ODP_UpdateConfigArea, ST *)
FUNCTION ODP_UpdateConfigArea : BOOL
(* This function update the "ODP-Conf"-Area.
	|Index  | Content 	   	         | Description
	|-------|------------------------|-----------------------
	| 0.. 7 | PLC.StationId          | 
	| 8..10 | PLC.CurrentTime        | 
	|11..13 | PLC.StartTime          | 
	|14..16 | PLC.SyncTime           | 
	|  17   | Flag SetTime           | indicates that the local RTC should be set to SyncTime	 
	- Update "PLC.CurrentTime" each cycle.
	- Set local RTC with a given "PLC.SyncTime" when requested by "Flag SetTime". 	
	  After work is done the request flag will reset.
	|-------|------------------------|-----------------------
	|  18   | PLC.BuildNumber        | This CoDeSys library version
	|  19   | PLC.TestedOdpVersion   | Tested with ODP2.7(SP1)
	|  20   | PLC.SupportedFeature	 | Bit 0, 1 and 3  
	|-------|------------------------|-----------------------
	|   30  | PLC.HistRecIntervall   | 1 Minute (constant)
	|   31  | PLC.HistRecDuration    | 24 Hours (constant)
	|   36  | PLC.HistInvalidValue   | 16#0000 (default, can be overwrite)
	|   37  | PLC.HistBuffClear      | indicates that the history should be set to "PLC.HistInvalidValue"
	- Publish the HistRecInterval and duration.
	- Reset all existing historical data when requested by "PLC.HistBuffClear"	  
	  After work is done the request flag will reset.
	  ===> This job is shift to program "ODP_AGENT", where all values of each histical variable reset in a separat plc-cycle, 
		   to provide a constant cycletime, who are not depending on the number of historical variables
	|-------|------------------------|-----------------------
	|   40  | PLC.AlmSendDataSize    | 5 + Number of Compressed alarmwords
	|50..52 | PLC.AlmLastAlarmTime   | Zero if no alarm detected
	|   53  | PLC.AlmLastAlarmID     | 16#0000 (constant)
	|   54  | PLC.AlmLastAlarmValue  | 16#0000 (constant)
	|   60  | PLC.AlmBuffClear       | Indicates that the alarmbuffer should be reset to zero
	|   61  | PLC.AlmResetSendTiming | IGNORED: send timing handled internaly by plc program 
	|   62  | PLC.AlmBuffSimulation  | IGNORED: not implemented
	|-------|------------------------|-----------------------
	|   63	| PLC.AlmBuffSendNow	 | Request flag for retransmission of AlmBuff (Flanke 0/1)
	- After work is done the request flag will resetet by plc.
	|-------|------------------------|-----------------------
	|   70  | PLC.AlmPointerAlarm    | "Alarmzeiger" in Alarm ringbuffer
	|   71  | PLC.AlmPointerSend     | "Sendezeiger" in Alarm ringbuffer
	|   72  | PLC.AlmTelegramInc     | "Telegramm Inkrementor" 
	|   80  | PLC.AlmSendIntervall   | t#1s   (constant): send timing handled internaly by plc program 
	|   81  | PLC.AlmSendReplyTimeOut| t#15s  (constant): send timing handled internaly by plc program
	|   82  | PLC.AlmSendRetries     | 0 (constant): Alarms will retransmit infinite 
	|   83  | PLC.AlmDelayTime1      | t#30s  (constant): 
	|   84  | PLC.AlmDelayTime2      | t#60s  (constant):
	|   85  | PLC.AlmDelayTime3      | t#120s (constant):
	|   86  | PLC.AlmDelayTime4      | t#240s (constant):
	|   87  | PLC.AlmDelayTime5      | t#480s (constant):
*)
VAR_INPUT
END_VAR
VAR
	(* Set local RTC  *)
	pstSyncTime : POINTER TO tODP_Time;
	dtSyncTime : DT; (* Seconds sins 01.01.1970 *)

	(* Update CurrentTime in ODP-Config block *)
	tCurrentTime : tODP_Time;
	pabHelp : POINTER TO ARRAY [0..13] OF BYTE;

	(* Little helpers *)
	wHelp : WORD;
	i : INT;
END_VAR
(* Check SetTime flag *)
IF gODP_awData[17] = 16#0001 THEN
	pstSyncTime := ADR(gODP_awData[14]);	(* Assign Pointer to SyncTime *)
	dtSyncTime := ODP_Time2DT(pstSyncTime^);(* Convert tODP_Time into DT *)
	SysRtcSetTime(dtSyncTime); 				(* Set local RTC  *)
	gODP_awData[17] := 16#0000; 			(* Reset SetTime Flag in ODP-Config block *)
END_IF;

(* Read CurrentTime *)
tCurrentTime := ODP_GetTime();
(* Set PLC_CurrentTime at index 8 *)
pabHelp := ADR(tCurrentTime);
FOR i:=0 TO 2 DO
	gODP_awData[8 +i] := SHL(BYTE_TO_WORD(pabHelp^[(2*i)+1]), 8) OR BYTE_TO_WORD(pabHelp^[(2*i)]);
END_FOR


gODP_awData[18] := 5;   (* "PLC.BuildNumber" (local CoDeSys library version) *)
gODP_awData[19] := 27;  (* "PLC.TestedOdpVersion"  *)
gODP_awData[20] := 11;  (* "PLC.SupportedFeature": 	Bit 0, 1 and 3 *)

(* Publish "HistRecInterval" and "HistRecDuration" *)
gODP_awData[30] := 60;  (* PLC.HistRecIntervall:  1 Minute (constant) *)
gODP_awData[31] := 1440;(* PLC.HistRecDuration:  24 Hours  (constant) *)

gODP_awData[36] := 65535;(* PLC.HistInvalidValue: *)
(* Publish "AlmSendDataSize" *)
gODP_awData[40] := UINT_TO_WORD(5 + gcODP_uiSIZE_COMPRESSEDALARMS);  (* 5 + Number of Compressed alarmwords *)

(* Publish "AlmLastAlarmTime" *)
pabHelp := ADR(grODP_asAlarmSendBuffer[grODP_uiCurrentAlarms].tTime);
FOR i:=0 TO 2 DO
	gODP_awData[50 +i] := SHL(BYTE_TO_WORD(pabHelp^[(2*i)+1]), 8) OR BYTE_TO_WORD(pabHelp^[(2*i)]);
END_FOR

(* Check if the alarmbuffer should be reset to zero *)
IF gODP_awData[60] = 16#0001 THEN
	pabHelp := ADR(grODP_asAlarmSendBuffer);
	FOR i:=0 TO SIZEOF(grODP_asAlarmSendBuffer)-1 DO
		pabHelp^[i] := 16#00;
	END_FOR
	grODP_uiCurrentAlarms := 16#00;
	grODP_uiTransmittedAlarms := 16#00;
	gODP_awData[60] := 16#0000; (* Reset Flag *)
END_IF

gODP_awData[70] := UINT_TO_WORD(grODP_uiCurrentAlarms); (* Publish "AlmPointerAlarm" *)
gODP_awData[71] := UINT_TO_WORD(grODP_uiTransmittedAlarms); (* Publish "AlmPointerSend" *)
gODP_awData[72] := UINT_TO_WORD(grODP_uiAlarmIncrementor); (* Publish "AlmTelegramInc" *)
gODP_awData[80] := 1;   (* Publish "AlmSendIntervall" *)
gODP_awData[81] := 15;  (* Publish "AlmSendReplyTimeOut" *)
gODP_awData[82] := 0;   (* Publish "AlmSendRetries" *)
gODP_awData[83] := 30;  (* Publish "AlmDelayTime1" *)
gODP_awData[84] := 60;  (* Publish "AlmDelayTime2" *)
gODP_awData[85] := 120; (* Publish "AlmDelayTime3" *)
gODP_awData[86] := 240; (* Publish "AlmDelayTime4" *)
gODP_awData[87] := 480; (* Publish "AlmDelayTime5" *)
END_FUNCTION

(* POU ODP_Time2DT, ST *)
FUNCTION ODP_Time2DT : DT
(* This function converts the memory friendly ODP format into IEC DT type (DT#yyyy-mm-dd-HH:MM.SS *)
VAR_INPUT
	 stT : tODP_Time;
END_VAR
VAR
	abTime : ARRAY [0..25] OF BYTE;
	psTime : POINTER TO STRING(25);
	sHelp : STRING;
	pabHelp : POINTER TO ARRAY [0..5] OF BYTE;
END_VAR
(* This function converts the memory friendly format into a readable string dt#1972-03-29-00:00:00 *)
(* Prefix *)
abTime[0] := 16#44; (* <D> *)
abTime[1] := 16#54; (* <T> *)
abTime[2] := 16#23; (* <#> *)
(* Year *)
sHelp := WORD_TO_STRING(BYTE_TO_WORD(stT.bYear) + 2000);
pabHelp := ADR(sHelp);
abTime[3] := pabHelp^[0];
abTime[4] := pabHelp^[1];
abTime[5] := pabHelp^[2];
abTime[6] := pabHelp^[3];
abTime[7] := 16#2D; (* <-> *)
(* Month *)
IF stT.bMonth <= 9 THEN
	abTime[8] := 16#30;
	abTime[9] := 16#30 + stT.bMonth;
ELSE
	sHelp := BYTE_TO_STRING(stT.bMonth);
	pabHelp := ADR(sHelp);
	abTime[8] := pabHelp^[0];
	abTime[9] := pabHelp^[1];
END_IF
abTime[10] := 16#2D; (* <-> *)
(* Day *)
IF stT.bDay <= 9 THEN
	abTime[11] := 16#30;
	abTime[12] := 16#30 + stT.bDay;
ELSE
	sHelp := BYTE_TO_STRING(stT.bDay);
	pabHelp := ADR(sHelp);
	abTime[11] := pabHelp^[0];
	abTime[12] := pabHelp^[1];
END_IF
abTime[13] := 16#2D; (* <-> *)
(* Hour *)
IF stT.bHour <= 9 THEN
	abTime[14] := 16#30;
	abTime[15] := 16#30 + stT.bHour;
ELSE
	sHelp := BYTE_TO_STRING(stT.bHour);
	pabHelp := ADR(sHelp);
	abTime[14] := pabHelp^[0];
	abTime[15] := pabHelp^[1];
END_IF
abTime[16] := 16#3A; (* <:> *)
(* Minute *)
IF stT.bMinute <= 9 THEN
	abTime[17] := 16#30;
	abTime[18] := 16#30 + stT.bMinute;
ELSE
	sHelp := BYTE_TO_STRING(stT.bMinute);
	pabHelp := ADR(sHelp);
	abTime[17] := pabHelp^[0];
	abTime[18] := pabHelp^[1];
END_IF
abTime[19] := 16#3A; (* <:> *)
(* Second *)
IF stT.bSecond <= 9 THEN
	abTime[20] := 16#30;
	abTime[21] := 16#30 + stT.bSecond;
ELSE
	sHelp := BYTE_TO_STRING(stT.bSecond);
	pabHelp := ADR(sHelp);
	abTime[20] := pabHelp^[0];
	abTime[21] := pabHelp^[1];
END_IF
abTime[22] := 16#00; (* [END] *)

psTime := ADR(abTime);
ODP_Time2DT := STRING_TO_DT(psTime^);
END_FUNCTION

(* POU ODP_CheckAlarms, ST *)
FUNCTION ODP_CheckAlarms : WORD
(* This function iterate through all configurated alarms and check current value of assoziated variable.
   In addition it set/reset the correspondent bit in the compressed repraesentaion 'gODP_awCompressedAlarms' 
	wReturn values:
		16#0000 ==> SUCCESS: Nothing to do
		16#0001 ==> ALARM DETECTED: Send modbus request to PC-Software "ODP-Config" 
*)
VAR_INPUT
	tCurTime : tODP_Time;
END_VAR
VAR
	wReturn : WORD;

	pxCurrentValue : POINTER TO BOOL;
	xCurrentValue : BOOL;
	(* Position of bit in compressed repraesentation 'gODP_awCompressedAlarms' *)
	wWordIndex : WORD;
	bBitIndex : BYTE;

	wHelp : WORD;
	i : INT;
END_VAR
wReturn := 16#0000; (* Init with SUCCESS *)

(* Check each alarm if state has changed *)
FOR i:=0 TO gODP_iCountAlarms-1 DO
	pxCurrentValue := gODP_asConfigAlarms[i].dwAddress;
	xCurrentValue := pxCurrentValue^;
	IF xCurrentValue <> gODP_asConfigAlarms[i].xOldValue THEN
		gODP_asConfigAlarms[i].xOldValue := xCurrentValue;
		wReturn := 16#0001; (* ALARM DETECTED: Send modbus request to PC-Software "ODP-Config" *)
		(* Read position in compressed repraesentation from 'gODP_asConfigAlarms' *)
		wWordIndex := gODP_asConfigAlarms[i].wMbWordIdx;
		bBitIndex := gODP_asConfigAlarms[i].bMbBitIdx;
		(* Update bit in compressed repraesetation of all alarms *)
		IF xCurrentValue THEN
			gODP_asConfigAlarms[i].eAlarmState := eOdpAlarmCOME;
			(* Set bit in compressed repraesetation *)
			wHelp := 16#0001;
			gODP_awCompressedAlarms[wWordIndex] := gODP_awCompressedAlarms[wWordIndex] OR (SHL(wHelp, bBitIndex));
			(* Update alarmLog *)
			ODP_UpdateAlarmLog(	gODP_asConfigAlarms[i].iTagId,
								eOdpAlarmCOME,
								tCurTime);
		ELSE
			gODP_asConfigAlarms[i].eAlarmState := eOdpAlarmGONE;
			(* Reset bit *)
			wHelp := 16#FFFE;
			wHelp := ROL(wHelp, bBitIndex);
			gODP_awCompressedAlarms[wWordIndex] := gODP_awCompressedAlarms[wWordIndex] AND wHelp;
			(* Update alarmLog *)
			ODP_UpdateAlarmLog(	gODP_asConfigAlarms[i].iTagId,
								eOdpAlarmGONE,
								tCurTime);
		END_IF
	END_IF
END_FOR

(* Check for retransmission of current alarms, requested by ODP-Server *)
IF gODP_awData[63] = 16#0001 THEN
	wReturn := 16#0001;
	gODP_awData[63] := 16#0000; (* Reset Flag *)
END_IF

(* Add entry into raw alarm send buffer *)
IF (wReturn = 16#0001) THEN (* ALARM DETECTED: Add compresses representation of all alarms into Alarmbuffer and increment Alarmpointer *)
	(* Increment "Alarmzeiger" *)
	grODP_uiCurrentAlarms := (grODP_uiCurrentAlarms +1) MOD gcODP_uiMAXALARMLOGENTRIES;
	(* Copy bitcoded (compressed alarms into send buffer *)
	FOR i:=0 TO (gcODP_uiSIZE_COMPRESSEDALARMS -1) DO
		grODP_asAlarmSendBuffer[grODP_uiCurrentAlarms].awCompressedAlarms[i] := gODP_awCompressedAlarms[i];
	END_FOR
	(* Add a timestamp *)
	grODP_asAlarmSendBuffer[grODP_uiCurrentAlarms].tTime := tCurTime;
	(* Verhindern, das "Alarmzeiger" den "Sendezeiger" überholt *)
	IF grODP_uiCurrentAlarms = grODP_uiTransmittedAlarms THEN
		grODP_uiTransmittedAlarms := (grODP_uiTransmittedAlarms +1) MOD gcODP_uiMAXALARMLOGENTRIES;
	END_IF
END_IF

ODP_CheckAlarms := wReturn;
END_FUNCTION

(* POU ODP_UpdateAlarmLog, ST *)
FUNCTION ODP_UpdateAlarmLog : WORD
(* This function adds one entriy into the alarm log 'grODP_asAlarmLog' *)
VAR_INPUT
	iTagId : INT;
	eAlarmState : tODP_AlarmState;
	tTime : tODP_Time;
END_VAR
VAR
END_VAR
(* Write to log *)
grODP_asAlarmLog[grODP_uiAlarmLogIndex].iTagId := iTagId;
grODP_asAlarmLog[grODP_uiAlarmLogIndex].eAlarmState := eAlarmState;
grODP_asAlarmLog[grODP_uiAlarmLogIndex].tTime := tTime;
(* Set index to the next free entry *)
grODP_uiAlarmLogIndex := (grODP_uiAlarmLogIndex +1) MOD gcODP_uiMAXALARMLOGENTRIES;
END_FUNCTION

(* POU ODP_UpdateHistory, ST *)
FUNCTION ODP_UpdateHistory : WORD
VAR_INPUT
	tCurTime : tODP_Time;
END_VAR
VAR
	wReturn : WORD;

	wSubIndex: WORD; (* Sub index to store historic data *)

	piHelp : POINTER TO INT;
	puiHelp : POINTER TO UINT;

	i : INT;
END_VAR
wReturn := 16#0000; (* Init with SUCCESS *)

(* Calculate Index in 'gODP_awData', depending of current time *)
wSubIndex := (BYTE_TO_WORD(tCurTime.bHour) *60) + BYTE_TO_WORD(tCurTime.bMinute);

(* Iterate along all hist variables *)
FOR i:=0 TO gODP_iCountHistoryVars-1 DO

	CASE gODP_asConfigHistory[i].eDataType OF
	eOdpTypeBOOL :(* BOOLEAN *)
		wReturn := 16#0001; (* ERROR: Unsupported data type detected in 'ODP_UpdateHistory'*)
		EXIT;
	eOdpTypeCHAR, eOdpTypeINT8, eOdpTypeUINT8 :(* BYTE *)
		wReturn := 16#0001; (* ERROR: Unsupported data type detected in 'ODP_UpdateHistory'*)
		EXIT;
	eOdpTypeINT16 :(* INT *)
		piHelp := gODP_asConfigHistory[i].dwAddress; (* assign address of local variable *)
		gODP_awData[gODP_asConfigHistory[i].wIndex + wSubIndex] := piHelp^;
	eOdpTypeUINT16 :(* WORD; UINT *)
		puiHelp := gODP_asConfigHistory[i].dwAddress; (* assign address of local variable *)
		gODP_awData[gODP_asConfigHistory[i].wIndex + wSubIndex] := puiHelp^;
	eOdpTypeINT32 :(* DINT *)
		wReturn := 16#0001; (* ERROR: Unsupported data type detected in 'ODP_UpdateHistory'*)
		EXIT;
	eOdpTypeUINT32 :(* DWORD; UDINT *)
		wReturn := 16#0001; (* ERROR: Unsupported data type detected in 'ODP_UpdateHistory'*)
		EXIT;
	eOdpTypeINT64 :(* QINT *)
		wReturn := 16#0001; (* ERROR: Unsupported data type detected in 'ODP_UpdateHistory'*)
		EXIT;
	eOdpTypeUINT64 :(* QWORD; UQINT *)
		wReturn := 16#0001; (* ERROR: Unsupported data type detected in 'ODP_UpdateHistory'*)
		EXIT;
	eOdpTypeFLOAT32 :(* REAL *)
		wReturn := 16#0001; (* ERROR: Unsupported data type detected in 'ODP_UpdateHistory'*)
		EXIT;
	eOdpTypeFLOAT64 :(* LREAL *)
		wReturn := 16#0001; (* ERROR: Unsupported data type detected in 'ODP_UpdateHistory'*)
		EXIT;
	eOdpTypeSTRING :(* String(230) *)
		wReturn := 16#0001; (* ERROR: Unsupported data type detected in 'ODP_UpdateHistory'*)
		EXIT;
	eOdpTypeBLOB :(* Binary Large OBject (max 230) *)
		wReturn := 16#0001; (* ERROR: Unsupported data type detected in 'ODP_UpdateHistory'*)
		EXIT;
	ELSE
		wReturn := 16#0001; (* ERROR: Unsupported data type detected in 'ODP_UpdateHistory'*)
	END_CASE
END_FOR

ODP_UpdateHistory := wReturn;
END_FUNCTION

(* POU ODP_UpdateOnlineWriteArea, ST *)
FUNCTION ODP_UpdateOnlineWriteArea : WORD
(* This function updates lokale variables with values written by PC-Software "ODP-Config".
	wReturn values:
		16#0000 ==> SUCCESS
		16#0001 ==> ERROR: Unsupported data type detected
*)
VAR_INPUT
END_VAR
VAR
	wReturn : WORD;

	puiHelp : POINTER TO UINT;
	piHelp : POINTER TO INT;

	i : INT;
END_VAR
wReturn := 16#0000; (* Init with SUCCESS *)

FOR i:=0 TO gODP_iCountOnlineWriteVars-1 DO
	CASE gODP_asConfigWrite[i].eDataType OF
	eOdpTypeBOOL :(* BOOLEAN *)
		wReturn := 16#0001; (* ERROR: Unsupported data type detected in 'ODP_UpdateOnlineWriteArea'*)
		EXIT;
	eOdpTypeCHAR, eOdpTypeINT8, eOdpTypeUINT8 :(* BYTE *)
		wReturn := 16#0001; (* ERROR: Unsupported data type detected in 'ODP_UpdateOnlineWriteArea'*)
		EXIT;
	eOdpTypeINT16 :(* INT *)
		piHelp := gODP_asConfigWrite[i].dwAddress; (* assign address of local variable *)
		piHelp^:= gODP_awData[gODP_asConfigWrite[i].wIndex];
	eOdpTypeUINT16 :(* WORD; UINT *)
		puiHelp := gODP_asConfigWrite[i].dwAddress; (* assign address of local variable *)
		puiHelp^:= gODP_awData[gODP_asConfigWrite[i].wIndex];
	eOdpTypeINT32 :(* DINT *)
		wReturn := 16#0001; (* ERROR: Unsupported data type detected in 'ODP_UpdateOnlineWriteArea'*)
		EXIT;
	eOdpTypeUINT32 :(* DWORD; UDINT *)
		wReturn := 16#0001; (* ERROR: Unsupported data type detected in 'ODP_UpdateOnlineWriteArea'*)
		EXIT;
	eOdpTypeINT64 :(* QINT *)
		wReturn := 16#0001; (* ERROR: Unsupported data type detected in 'ODP_UpdateOnlineWriteArea'*)
		EXIT;
	eOdpTypeUINT64 :(* QWORD; UQINT *)
		wReturn := 16#0001; (* ERROR: Unsupported data type detected in 'ODP_UpdateOnlineWriteArea'*)
		EXIT;
	eOdpTypeFLOAT32 :(* REAL *)
		wReturn := 16#0001; (* ERROR: Unsupported data type detected in 'ODP_UpdateOnlineWriteArea'*)
		EXIT;
	eOdpTypeFLOAT64 :(* LREAL *)
		wReturn := 16#0001; (* ERROR: Unsupported data type detected in 'ODP_UpdateOnlineWriteArea'*)
		EXIT;
	eOdpTypeSTRING :(* String(230) *)
		wReturn := 16#0001; (* ERROR: Unsupported data type detected in 'ODP_UpdateOnlineWriteArea'*)
		EXIT;
	eOdpTypeBLOB :(* Binary Large OBject (max 230) *)
		wReturn := 16#0001; (* ERROR: Unsupported data type detected in 'ODP_UpdateOnlineWriteArea'*)
		EXIT;
	ELSE
		wReturn := 16#0001; (* ERROR: Unsupported data type detected in 'ODP_UpdateOnlineWriteArea'*)
	END_CASE
END_FOR

ODP_UpdateOnlineWriteArea := wReturn;
END_FUNCTION

(* POU ODP_UpdateOnlineReadArea, ST *)
FUNCTION ODP_UpdateOnlineReadArea : WORD
(* This function updates the OnlineReadArea with values of lokale variables.
   In addition it calls 'ODP_UpdateRTC()'.  
   The OnlineReadArea will be readed cycled by PC-Software "ODP-Config".
	wReturn values:
		16#0000 ==> SUCCESS
		16#0001 ==> ERROR: Unsupported data type detected
*)
VAR_INPUT
END_VAR
VAR
	wReturn : WORD;

	piHelp : POINTER TO INT;
	puiHelp : POINTER TO UINT;

	i : INT;
END_VAR
wReturn := 16#0000; (* Init with SUCCESS *)

FOR i:=0 TO gODP_iCountOnlineReadVars-1 DO
	CASE gODP_asConfigRead[i].eDataType OF
	eOdpTypeBOOL :(* BOOLEAN *)
		wReturn := 16#0001; (* ERROR: Unsupported data type detected in 'ODP_UpdateOnlineReadArea'*)
		EXIT;
	eOdpTypeCHAR, eOdpTypeINT8, eOdpTypeUINT8 :(* BYTE *)
		wReturn := 16#0001; (* ERROR: Unsupported data type detected in 'ODP_UpdateOnlineReadArea'*)
		EXIT;
	eOdpTypeINT16 :(* INT *)
		piHelp := gODP_asConfigRead[i].dwAddress; (* assign address of local variable *)
		gODP_awData[gODP_asConfigRead[i].wIndex] := piHelp^;
	eOdpTypeUINT16 :(* WORD; UINT *)
		puiHelp := gODP_asConfigRead[i].dwAddress; (* assign address of local variable *)
		gODP_awData[gODP_asConfigRead[i].wIndex] := puiHelp^;
	eOdpTypeINT32 :(* DINT *)
		wReturn := 16#0001; (* ERROR: Unsupported data type detected in 'ODP_UpdateOnlineReadArea'*)
		EXIT;
	eOdpTypeUINT32 :(* DWORD; UDINT *)
		wReturn := 16#0001; (* ERROR: Unsupported data type detected in 'ODP_UpdateOnlineReadArea'*)
		EXIT;
	eOdpTypeINT64 :(* QINT *)
		wReturn := 16#0001; (* ERROR: Unsupported data type detected in 'ODP_UpdateOnlineReadArea'*)
		EXIT;
	eOdpTypeUINT64 :(* QWORD; UQINT *)
		wReturn := 16#0001; (* ERROR: Unsupported data type detected in 'ODP_UpdateOnlineReadArea'*)
		EXIT;
	eOdpTypeFLOAT32 :(* REAL *)
		wReturn := 16#0001; (* ERROR: Unsupported data type detected in 'ODP_UpdateOnlineReadArea'*)
		EXIT;
	eOdpTypeFLOAT64 :(* LREAL *)
		wReturn := 16#0001; (* ERROR: Unsupported data type detected in 'ODP_UpdateOnlineReadArea'*)
		EXIT;
	eOdpTypeSTRING :(* String(230) *)
		wReturn := 16#0001; (* ERROR: Unsupported data type detected in 'ODP_UpdateOnlineReadArea'*)
		EXIT;
	eOdpTypeBLOB :(* Binary Large OBject (max 230) *)
		wReturn := 16#0001; (* ERROR: Unsupported data type detected in 'ODP_UpdateOnlineReadArea'*)
		EXIT;
	ELSE
		wReturn := 16#0001; (* ERROR: Unsupported data type detected in 'ODP_UpdateOnlineReadArea'*)
	END_CASE
END_FOR

ODP_UpdateOnlineReadArea := wReturn;
END_FUNCTION

(* POU ODP_InitOdpConfig, ST *)
FUNCTION ODP_InitOdpConfig : BOOL
(* This function set in ODP-Config block the:
   - StationID 								(at index 0).
   - UpdateIntervall for OnlineReadArea.
   - PlcStartTime 							(at index 11).
   - PlcCurrentTime(init)  					(at index 8). 
   - ...
	Return values:
		TRUE  ==> SUCCESS
		FALSE ==> ERROR
*)
VAR_INPUT
	sStationId : STRING(14);
	tOnlineIntervall : TIME;
END_VAR
VAR
	tOdpTime : tODP_Time;
	pabHelp : POINTER TO ARRAY [0..15] OF BYTE;
	i : INT;
END_VAR
(* Set StationID *)
pabHelp := ADR(sStationId);
FOR i:=0 TO 7 DO
	gODP_awData[i] := SHL(BYTE_TO_WORD(pabHelp^[(2*i)+1]), 8) OR BYTE_TO_WORD(pabHelp^[(2*i)]);
END_FOR
(* Set Intervall to update the OnlineReadArea *)
gODP_tOnlineIntervall := tOnlineIntervall;

(* Read CurrentTime  *)
tOdpTime := ODP_GetTime();
(* Set PLC_CurrentTime at index 8 *)
pabHelp := ADR(tOdpTime);
FOR i:=0 TO 2 DO
	gODP_awData[8 +i] := SHL(BYTE_TO_WORD(pabHelp^[(2*i)+1]), 8) OR BYTE_TO_WORD(pabHelp^[(2*i)]);
END_FOR
(* Set PLC_StartTime at index 11 *)
pabHelp := ADR(tOdpTime);
FOR i:=0 TO 2 DO
	gODP_awData[11 +i] := SHL(BYTE_TO_WORD(pabHelp^[(2*i)+1]), 8) OR BYTE_TO_WORD(pabHelp^[(2*i)]);
END_FOR
END_FUNCTION

(* POU ODP_RegisterTag, ST *)
FUNCTION ODP_RegisterTag : WORD
(* This function add a variable to the list of monitored variables.
	Return values:
		16#0000 ==> SUCCESS
		16#0001 ==> ERROR: Unknown ODP-Table
		16#0002 ==> ERROR: TagName to long, max 12 Char
		16#0003 ==> ERROR: No more memory for additional tag's
		16#0004 ==> ERROR: Maximum number of variables are configuraed in specified table.  
		16#0005 ==> ERROR: Alarms must be of type BOOL.
		16#0006 ==> ERROR: No more memory for additional tag's in historyarea. It will overlapp the AlarmArea. 
  
*)
VAR_INPUT
	eOdpTable: tODP_Table;		(* eOdpOnlineRead, eOdpOnlineWrite, eOdpHistory or eOdpAlarm *)
	sTagName : STRING(12); 		(* TagName, displayed in ODP-Config *)
	dwAddress: DWORD; 			(* Address of variable that should be monitored *)
	eOdpType : tODP_DataType;	(* DataType of variable *)
END_VAR
VAR
	wReturn : WORD;
	wHelp : WORD;
END_VAR
wReturn := 16#0000; (* Init with SUCCESS *)

CASE eOdpTable OF
eOdpTableRead : (* Add to OnlineReadArea *)
	IF gODP_iCountOnlineReadVars +1 >= gcODP_uiMAXVAR_ONLINEREAD THEN
		wReturn := 16#0004; (* ERROR: Maximum number of variables are configuraed in specified table *)
	ELSE
		gODP_asConfigRead[gODP_iCountOnlineReadVars].sTagName  := sTagName;
		gODP_asConfigRead[gODP_iCountOnlineReadVars].dwAddress := dwAddress;
		gODP_asConfigRead[gODP_iCountOnlineReadVars].eDataType := eOdpType;
		IF gODP_iCountOnlineReadVars = 0 THEN
			gODP_asConfigRead[gODP_iCountOnlineReadVars].wIndex := gcODP_uiOFFSET_ONLINEREAD;
		ELSE
			wHelp := gODP_asConfigRead[gODP_iCountOnlineReadVars-1].wIndex; (* Get Index of last variable *)
			wHelp := wHelp + ODP_SizeOfOdpDataType(gODP_asConfigRead[gODP_iCountOnlineReadVars-1].eDataType);
			gODP_asConfigRead[gODP_iCountOnlineReadVars].wIndex := wHelp;
		END_IF
		gODP_iCountOnlineReadVars := gODP_iCountOnlineReadVars +1;
	END_IF

eOdpTableWrite: (* Add to OnlineWriteArea *)
	IF gODP_iCountOnlineWriteVars +1 >= gcODP_uiMAXVAR_ONLINEWRITE THEN
		wReturn := 16#0004; (* ERROR: Maximum number of variables are configuraed in specified table *)
	ELSE
		gODP_asConfigWrite[gODP_iCountOnlineWriteVars].sTagName  := sTagName;
		gODP_asConfigWrite[gODP_iCountOnlineWriteVars].dwAddress := dwAddress;
		gODP_asConfigWrite[gODP_iCountOnlineWriteVars].eDataType := eOdpType;
		IF gODP_iCountOnlineWriteVars = 0 THEN
			gODP_asConfigWrite[gODP_iCountOnlineWriteVars].wIndex := gcODP_uiOFFSET_ONLINEWRITE;
		ELSE
			wHelp := gODP_asConfigWrite[gODP_iCountOnlineWriteVars-1].wIndex; (* Get Index of last variable *)
			wHelp := wHelp + ODP_SizeOfOdpDataType(gODP_asConfigWrite[gODP_iCountOnlineWriteVars-1].eDataType);
			gODP_asConfigWrite[gODP_iCountOnlineWriteVars].wIndex := wHelp;
		END_IF
		gODP_iCountOnlineWriteVars := gODP_iCountOnlineWriteVars +1;
	END_IF

eOdpTableHistory: (* Add to HistoryArea *)
	IF gODP_iCountHistoryVars +1 >= gcODP_uiMAXVAR_HISTORY THEN
		wReturn := 16#0004; (* ERROR: Maximum number of variables are configuraed in specified table *)
	ELSE
		gODP_asConfigHistory[gODP_iCountHistoryVars].sTagName  := sTagName;
		gODP_asConfigHistory[gODP_iCountHistoryVars].dwAddress := dwAddress;
		gODP_asConfigHistory[gODP_iCountHistoryVars].eDataType := eOdpType;
		(* Calculate startaddress of item in modbus buffer *)
		wHelp := gcODP_uiOFFSET_HISTORY_BASE + (gODP_iCountHistoryVars * gcODP_uiHISTORY_ITEM_SIZE);
		IF (wHelp + gcODP_uiHISTORY_ITEM_SIZE) >= gcODP_uiOFFSET_ALARM THEN
			wReturn := 16#0006; (* ERROR: No more memory FOR additional tag's in historyarea. It will overlapp the AlarmArea.*)
		ELSE
			gODP_asConfigHistory[gODP_iCountHistoryVars].wIndex := wHelp;
			(* Increment Counter of registerd HistoryVars *)
			gODP_iCountHistoryVars := gODP_iCountHistoryVars +1;
		END_IF
	END_IF

eOdpTableAlarm: (* Add to AlarmArea *)
	IF gODP_iCountAlarms +1 >= gcODP_uiMAXVAR_ALARMS THEN
		wReturn := 16#0004; (* ERROR: Maximum number of variables are configuraed in specified table *)
	ELSE
		IF eOdpType <> eOdpTypeBOOL THEN
			wReturn := 16#0005; (* ERROR: Alarms must be of type BOOL *)
		ELSE
			gODP_asConfigAlarms[gODP_iCountAlarms].sTagName  := sTagName;
			gODP_asConfigAlarms[gODP_iCountAlarms].iTagId    := gODP_iCountAlarms;
			gODP_asConfigAlarms[gODP_iCountAlarms].dwAddress := dwAddress;
			(* Calculate Word and Bit address of item in modbus buffer *)
			gODP_asConfigAlarms[gODP_iCountAlarms].wMbWordIdx := gODP_iCountAlarms/16;
			gODP_asConfigAlarms[gODP_iCountAlarms].bMbBitIdx := INT_TO_BYTE(gODP_iCountAlarms MOD 16);
			(* Increment Counter of registerd Alarms *)
			gODP_iCountAlarms := gODP_iCountAlarms +1;
		END_IF
	END_IF
ELSE
	wReturn := 16#0001; (* ERROR: Unknown ODP-Table *)
END_CASE

ODP_RegisterTag := wReturn;
END_FUNCTION

(* POU ODP_SizeOfOdpDataType, ST *)
FUNCTION ODP_SizeOfOdpDataType : WORD
(* This function returns the size in "WORD" of the given tODP_DataType *)
VAR_INPUT
	eOdpType : tODP_DataType;	(* DataType of variable *)
END_VAR
VAR
END_VAR
CASE eOdpType OF
  eOdpTypeBOOL, eOdpTypeCHAR, eOdpTypeINT8, eOdpTypeUINT8, eOdpTypeINT16, eOdpTypeUINT16:
	ODP_SizeOfOdpDataType := 1;
  eOdpTypeINT32, eOdpTypeUINT32, eOdpTypeFLOAT32:
	ODP_SizeOfOdpDataType := 2;
  eOdpTypeINT64, eOdpTypeUINT64, eOdpTypeFLOAT64:
	ODP_SizeOfOdpDataType := 4;
  eOdpTypeSTRING, eOdpTypeBLOB:
	ODP_SizeOfOdpDataType := 230;
END_CASE
END_FUNCTION

(* POU ODP_Time2String, ST *)
FUNCTION ODP_Time2String : STRING(25)
(* This function converts the memory friendly format into a readable string "dd.mm.yyyy HH:MM.SS" *)
VAR_INPUT
	 stT : tODP_Time;
END_VAR
VAR
	abTime : ARRAY [0..25] OF BYTE;
	psTime : POINTER TO STRING(25);
	sHelp : STRING;
	pabHelp : POINTER TO ARRAY [0..5] OF BYTE;
END_VAR
(* This function converts the memory friendly format into a readable string "dd.mm.yyyy HH:MM.SS" *)

(* Day *)
IF stT.bDay <= 9 THEN
	abTime[0] := 16#30;
	abTime[1] := 16#30 + stT.bDay;
ELSE
	sHelp := BYTE_TO_STRING(stT.bDay);
	pabHelp := ADR(sHelp);
	abTime[0] := pabHelp^[0];
	abTime[1] := pabHelp^[1];
END_IF
abTime[2] := 16#2E; (* . *)
(* Month *)
IF stT.bMonth <= 9 THEN
	abTime[3] := 16#30;
	abTime[4] := 16#30 + stT.bMonth;
ELSE
	sHelp := BYTE_TO_STRING(stT.bMonth);
	pabHelp := ADR(sHelp);
	abTime[3] := pabHelp^[0];
	abTime[4] := pabHelp^[1];
END_IF
abTime[5] := 16#2E; (* . *)
(* Year *)
sHelp := WORD_TO_STRING(BYTE_TO_WORD(stT.bYear) + 2000);
pabHelp := ADR(sHelp);
abTime[6] := pabHelp^[0];
abTime[7] := pabHelp^[1];
abTime[8] := pabHelp^[2];
abTime[9] := pabHelp^[3];
abTime[10] := 16#20; (* [SPACE] *)
(* Hour *)
IF stT.bHour <= 9 THEN
	abTime[11] := 16#30;
	abTime[12] := 16#30 + stT.bHour;
ELSE
	sHelp := BYTE_TO_STRING(stT.bHour);
	pabHelp := ADR(sHelp);
	abTime[11] := pabHelp^[0];
	abTime[12] := pabHelp^[1];
END_IF
abTime[13] := 16#3A; (* : *)
(* Minute *)
IF stT.bMinute <= 9 THEN
	abTime[14] := 16#30;
	abTime[15] := 16#30 + stT.bMinute;
ELSE
	sHelp := BYTE_TO_STRING(stT.bMinute);
	pabHelp := ADR(sHelp);
	abTime[14] := pabHelp^[0];
	abTime[15] := pabHelp^[1];
END_IF
abTime[16] := 16#3A; (* : *)
(* Second *)
IF stT.bSecond <= 9 THEN
	abTime[17] := 16#30;
	abTime[18] := 16#30 + stT.bSecond;
ELSE
	sHelp := BYTE_TO_STRING(stT.bSecond);
	pabHelp := ADR(sHelp);
	abTime[17] := pabHelp^[0];
	abTime[18] := pabHelp^[1];
END_IF
abTime[19] := 16#00; (* [END] *)

psTime := ADR(abTime);
ODP_Time2String := psTime^;
END_FUNCTION

(* POU ODP_VERSION, ST *)
FUNCTION ODP_VERSION : WORD
(*

 date     | release	| author  | Desc
----------+---------+------------------------------------------------------------
 07.03.08 |  1.0	| CM      | Init based on "ODP Specification 1.2 Rev.A"(restricted to 16 alarms)
 24.04.08 |  1.1    | CM      | Update alarmhandling to "ODP Specification 1.3 Rev.D"
 09.02.10 |  1.2    | CM/MJ	  | Interop-Test "WagoLibODP_02.lib" mit ODP-Server 2.7SP1
 29.03.10 |  1.3    | CM	  | Add "AlmBuffSendNow" feature
 09.06.10 |  1.4    | CM	  | Add "outputs" to ODP_AGENT for status information  
 10.06.10 |  1.5    | CM	  | Redesign of retransmission behaivior for alarms
 24.06.10 |  1.6    | CM	  | BugFix: ReceiveBuffer handling
 29.06.10 |  1.7    | CM	  | Add "Delay" between two transmissions 

 *)
VAR_INPUT
END_VAR
VAR
	(* Current library version *)
	bMajor : BYTE := 16#01;
	bMinor : BYTE := 16#07;
END_VAR
ODP_VERSION := SHL(BYTE_TO_WORD(bMajor), 8) OR BYTE_TO_WORD(bMinor);
END_FUNCTION
